FUNCTION_BLOCK FB2_Counters
VAR_INPUT
END_VAR
VAR_OUTPUT
END_VAR
VAR
	t_timerHigh : TON;
	t_timerLow : TP;
	b_eenHzClk : BOOL;
	b_eenHzTrigger : R_Trig;
	i_productieTimerSec: DINT;
	i_productieTimerMin: DINT;
	i_productieTimerHour: DINT;
END_VAR
VAR // added by the converter: edge detectors and wires of the graphical bodies
    _w1, _w2 : BOOL;
END_VAR

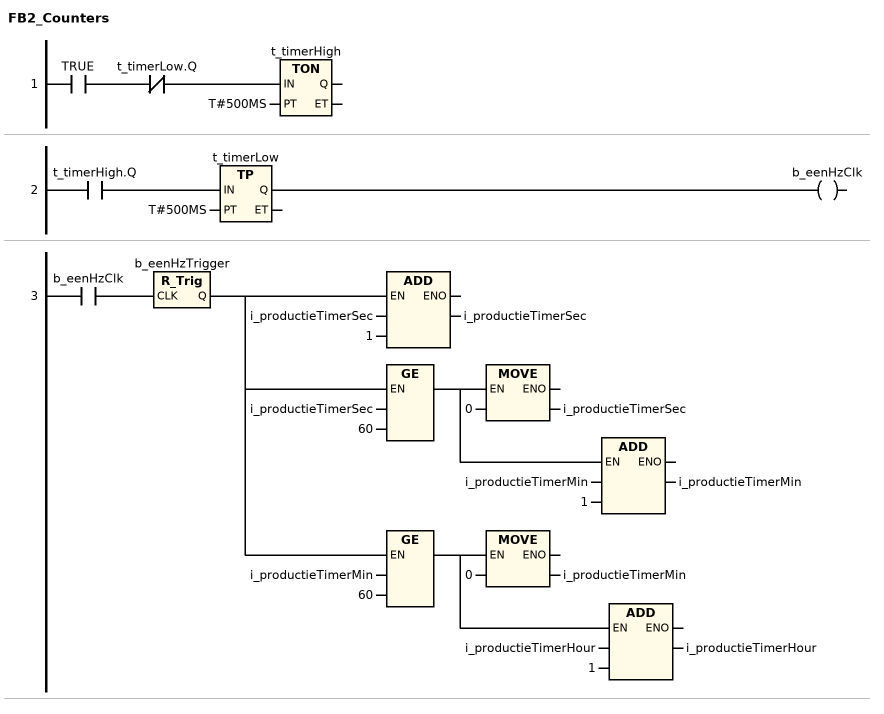
// NETWORK 1
t_timerHigh(IN := TRUE AND NOT t_timerLow.Q, PT := T#500MS); // TON

// NETWORK 2
t_timerLow(IN := t_timerHigh.Q, PT := T#500MS); // TP
b_eenHzClk := t_timerLow.Q;

// NETWORK 3
b_eenHzTrigger(CLK := b_eenHzClk); // R_Trig
IF b_eenHzTrigger.Q THEN i_productieTimerSec := i_productieTimerSec + 1; END_IF
_w1 := b_eenHzTrigger.Q AND i_productieTimerSec >= 60;
IF _w1 THEN i_productieTimerSec := 0; END_IF
IF _w1 THEN i_productieTimerMin := i_productieTimerMin + 1; END_IF
_w2 := b_eenHzTrigger.Q AND i_productieTimerMin >= 60;
IF _w2 THEN i_productieTimerMin := 0; END_IF
IF _w2 THEN i_productieTimerHour := i_productieTimerHour + 1; END_IF

END_FUNCTION_BLOCK

(* stored: Version 1.1.0.1, ProductVersion 3.1.4024.12
   POU FB2_Counters: Id {37e910bb-9530-4a49-ba25-fc8476665f5e}, SpecialFunc None *)
